{attribute wpf [Container(Layout.Wrap)]}
{attribute wpf [Group(Layout.GroupBox)]}
FUNCTION_BLOCK fbPneumaticActuator
VAR_INPUT
	{attribute wpf [Container(Layout.Stack)]}	
	{attribute addProperty Name "Retracted"}
	{attribute addProperty ToolTip "Sensor indicating that the actuator is retracted"}
	inRetracted : BOOL;	
	{attribute addProperty Name "Extend"}
	{attribute addProperty ToolTip "Sensor indicating that the actuator is extended"}
	inExtended : BOOL;	
END_VAR
VAR_OUTPUT
	{attribute wpf [Container(Layout.Stack)]}
	{attribute addProperty Name "Retract"}
	{attribute addProperty ToolTip "Signal for retracting"}
	outRetract : BOOL;
	{attribute addProperty Name "Extend"}
	{attribute addProperty ToolTip "Signal for Extending"}
	outExtend : BOOL;
END_VAR
VAR
	{attribute wpf [Container(Layout.UniformGrid)]}
	{attribute addProperty Name "Manual Retract"}
	{attribute addProperty ToolTip "Executes retraction in manual mode"}
	_manualRetract : BOOL;
	{attribute addProperty Name "Manual Extend"}
	{attribute addProperty ToolTip "Executes extension in manual mode"}
	_manualExtend : BOOL;
END_VAR

METHOD Extend : BOOL
THIS^.outRetract := FALSE;
THIS^.outExtend := TRUE;

Extend := THIS^.inExtended;
END_METHOD

METHOD Manual
IF(THIS^._manualExtend AND_THEN THIS^.Extend()) THEN THIS^._manualExtend := FALSE; END_IF;
IF(THIS^._manualRetract AND_THEN THIS^.Retract()) THEN THIS^._manualRetract := FALSE; END_IF;
END_METHOD

METHOD Retract : BOOL
THIS^.outRetract := TRUE;
THIS^.outExtend := FALSE;

Retract := THIS^.inRetracted;
END_METHOD

END_FUNCTION_BLOCK

(* stored: Version 1.1.0.1, ProductVersion 3.1.4024.3
   POU fbPneumaticActuator: Id {0897ab47-2dcc-4aaf-a97d-9b6927968f1d}, SpecialFunc None
   Method Extend: Id {4f8afd74-75b4-4631-a3c1-60b5d2b2c6d7}
   Method Manual: Id {e6a42619-97d5-4f12-a513-82a72cd35d49}
   Method Retract: Id {b1f8fc57-17ea-4721-8bb1-f5236524cc91} *)
